FUNCTION_BLOCK FB_Conveyor
VAR_INPUT
	Occupied	: BOOL;
	Takeover	: BOOL;
	Handover	: BOOL;
END_VAR
VAR_OUTPUT
	EnableMotor	: BOOL;
	Taking		: BOOL;
	Giving		: BOOL;
END_VAR
VAR
	transportState	: INT;
END_VAR


CASE transportState OF
	0:
	// Init
		Taking 		:= FALSE;
		Giving 		:= FALSE;
		EnableMotor := FALSE;
		transportState := 10;
	10:
	// Takeover or handover
		IF NOT Occupied THEN
			Taking 			:= TRUE;
			Giving 			:= FALSE;
			transportState 	:= 20;	
		ELSE
			Taking 			:= FALSE;
			Giving 			:= TRUE;
			transportState 	:= 200;
		END_IF
	20:
	// Takeover start
		IF Takeover THEN
			EnableMotor 	:= TRUE;
			transportState 	:= 21;
		END_IF		
	21:
	// Occupied
		IF Occupied THEN
			EnableMotor 	:= FALSE;
			Taking			:= FALSE;
			transportState 	:= 10;	
		END_IF		
	200:
	// Handover start
		IF Handover THEN
			Giving 			:= TRUE;
			EnableMotor 	:= TRUE;
			transportState 	:= 210;	
		END_IF
	210:
	// Handover completed
		IF NOT Occupied AND NOT Handover THEN
			EnableMotor		:= FALSE;
			Giving			:= FALSE;
			transportState 	:= 10;	
		END_IF
END_CASE

END_FUNCTION_BLOCK

(* stored: Version 1.1.0.1, ProductVersion 3.1.4022.18
   POU FB_Conveyor: Id {20a31204-5f1b-4ba7-95ba-c89133dce1b5}, SpecialFunc None *)
